% RSLogix 500 project TANK ANALOG CONTROL WITH ALARMS.RSS, saved by version 8.30.00.16 %
PROJECT "UNTITLED"    % processor: Bul.1763 MicroLogix 1100 Series B %

PROGRAM FILES
  LAD 2 "MAIN"  4 rungs
  LAD 3 "I/O"  5 rungs
  LAD 4 "CONTROLS"  6 rungs
  LAD 5 "ALARMS"  7 rungs

DATA FILES
  O0 OUTPUT  5 elements
  I1 INPUT  14 elements
  S2 STATUS  66 elements
  B3 BINARY  2 elements
  T4 TIMER  4 elements
  C5 COUNTER  1 elements
  R6 CONTROL  1 elements
  N7 INTEGER  1 elements
  F8 FLOAT  1 elements

LADDER 2 "MAIN"
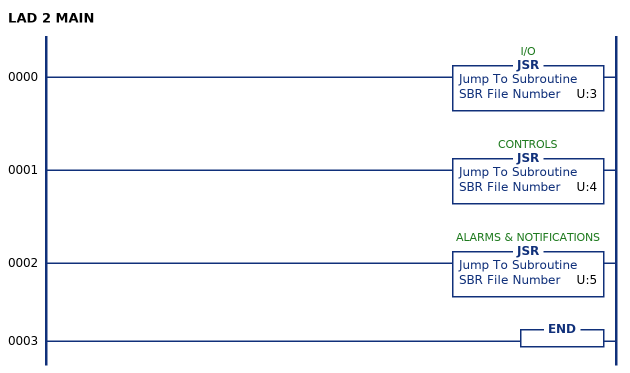
% Rung: 0 %
SOR JSR U:3 EOR
%   U:3  "I/O" %
% Rung: 1 %
SOR JSR U:4 EOR
%   U:4  "CONTROLS" %
% Rung: 2 %
SOR JSR U:5 EOR
%   U:5  "ALARMS & NOTIFICATIONS" %
% Rung: 3 %
SOR END EOR

LADDER 3 "I/O"
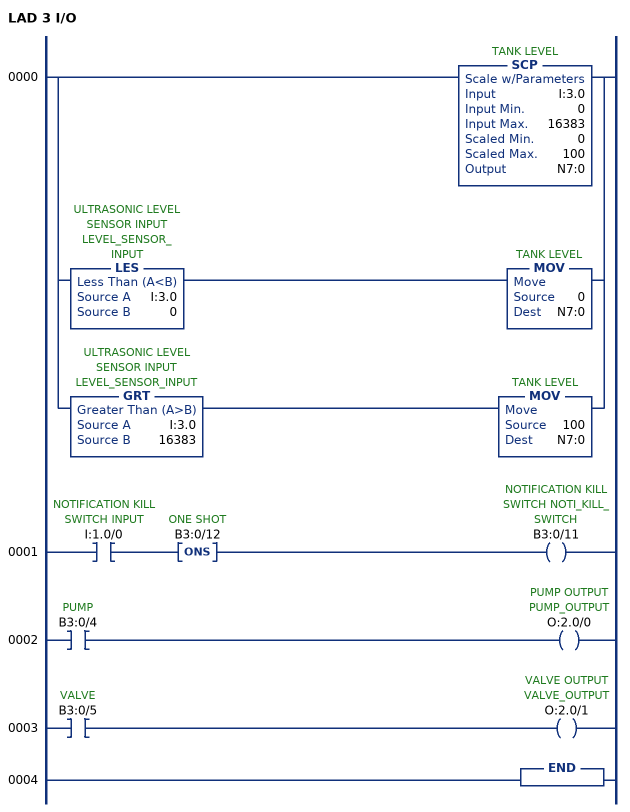
% Rung: 0 %
SOR BST SCP I:3.0 0 16383 0 100 N7:0 NXB LES I:3.0 0 MOV 0 N7:0 NXB GRT I:3.0 16383 MOV 100 N7:0 BND EOR
%   I:3.0  LEVEL_SENSOR_INPUT  "ULTRASONIC LEVEL SENSOR INPUT" %
%   N7:0  "TANK LEVEL" %
% Rung: 1 %
SOR XIC I:1.0/0 ONS B3:0/12 OTE B3:0/11 EOR
%   I:1.0/0  "NOTIFICATION KILL SWITCH INPUT" %
%   B3:0/12  "ONE SHOT" %
%   B3:0/11  NOTI_KILL_SWITCH  "NOTIFICATION KILL SWITCH" %
% Rung: 2 %
SOR XIC B3:0/4 OTE O:2.0/0 EOR
%   B3:0/4  "PUMP" %
%   O:2.0/0  PUMP_OUTPUT  "PUMP OUTPUT" %
% Rung: 3 %
SOR XIC B3:0/5 OTE O:2.0/1 EOR
%   B3:0/5  "VALVE" %
%   O:2.0/1  VALVE_OUTPUT  "VALVE OUTPUT" %
% Rung: 4 %
SOR END EOR

LADDER 4 "CONTROLS"
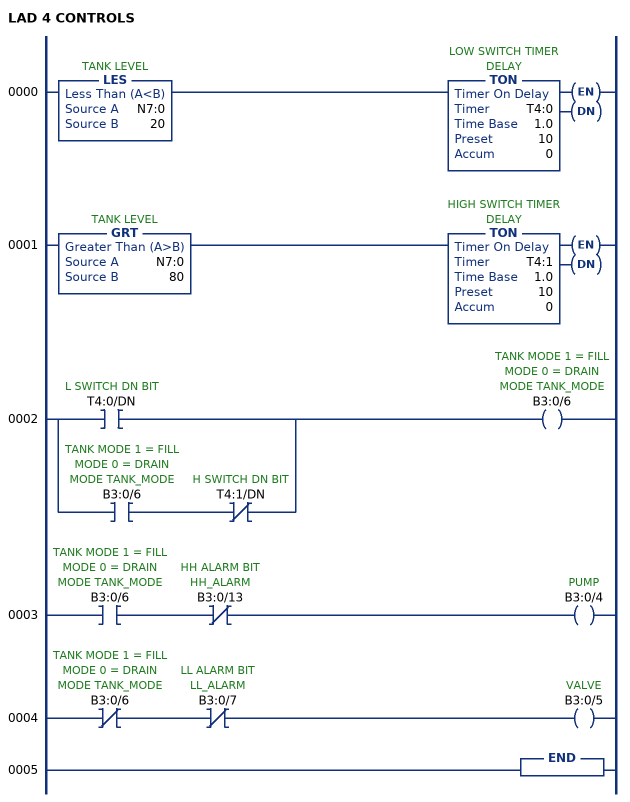
% Rung: 0 %
SOR LES N7:0 20 TON T4:0 1.0 10 0 EOR
%   N7:0  "TANK LEVEL" %
%   T4:0  "LOW SWITCH TIMER DELAY" %
% Rung: 1 %
SOR GRT N7:0 80 TON T4:1 1.0 10 0 EOR
%   N7:0  "TANK LEVEL" %
%   T4:1  "HIGH SWITCH TIMER DELAY" %
% Rung: 2 %
SOR BST XIC T4:0/DN NXB XIC B3:0/6 XIO T4:1/DN BND OTE B3:0/6 EOR
%   T4:0/DN  "L SWITCH DN BIT" %
%   B3:0/6  TANK_MODE  "TANK MODE 1 = FILL MODE 0 = DRAIN MODE" %
%   T4:1/DN  "H SWITCH DN BIT" %
% Rung: 3 %
SOR XIC B3:0/6 XIO B3:0/13 OTE B3:0/4 EOR
%   B3:0/6  TANK_MODE  "TANK MODE 1 = FILL MODE 0 = DRAIN MODE" %
%   B3:0/13  HH_ALARM  "HH ALARM BIT" %
%   B3:0/4  "PUMP" %
% Rung: 4 %
SOR XIO B3:0/6 XIO B3:0/7 OTE B3:0/5 EOR
%   B3:0/6  TANK_MODE  "TANK MODE 1 = FILL MODE 0 = DRAIN MODE" %
%   B3:0/7  LL_ALARM  "LL ALARM BIT" %
%   B3:0/5  "VALVE" %
% Rung: 5 %
SOR END EOR

LADDER 5 "ALARMS"
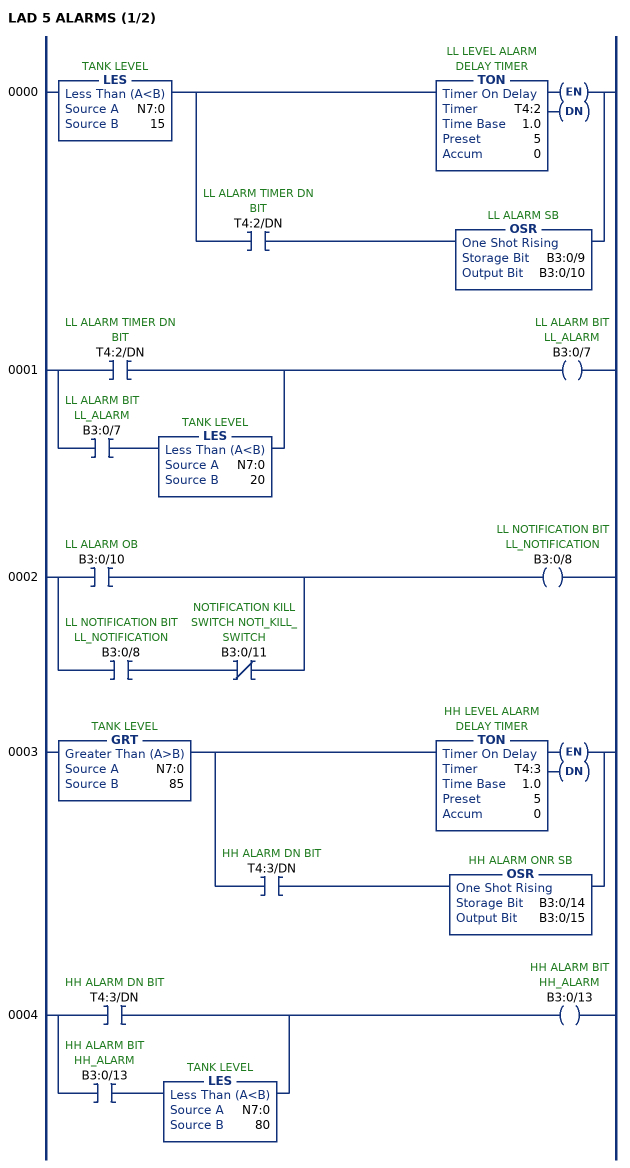
% Rung: 0 %
SOR LES N7:0 15 BST TON T4:2 1.0 5 0 NXB XIC T4:2/DN OSR B3:0/9 B3:0/10 BND EOR
%   N7:0  "TANK LEVEL" %
%   T4:2  "LL LEVEL ALARM DELAY TIMER" %
%   T4:2/DN  "LL ALARM TIMER DN BIT" %
%   B3:0/9  "LL ALARM SB" %
%   B3:0/10  "LL ALARM OB" %
% Rung: 1 %
SOR BST XIC T4:2/DN NXB XIC B3:0/7 LES N7:0 20 BND OTE B3:0/7 EOR
%   T4:2/DN  "LL ALARM TIMER DN BIT" %
%   B3:0/7  LL_ALARM  "LL ALARM BIT" %
%   N7:0  "TANK LEVEL" %
% Rung: 2 %
SOR BST XIC B3:0/10 NXB XIC B3:0/8 XIO B3:0/11 BND OTE B3:0/8 EOR
%   B3:0/10  "LL ALARM OB" %
%   B3:0/8  LL_NOTIFICATION  "LL NOTIFICATION BIT" %
%   B3:0/11  NOTI_KILL_SWITCH  "NOTIFICATION KILL SWITCH" %
% Rung: 3 %
SOR GRT N7:0 85 BST TON T4:3 1.0 5 0 NXB XIC T4:3/DN OSR B3:0/14 B3:0/15 BND EOR
%   N7:0  "TANK LEVEL" %
%   T4:3  "HH LEVEL ALARM DELAY TIMER" %
%   T4:3/DN  "HH ALARM DN BIT" %
%   B3:0/14  "HH ALARM ONR SB" %
%   B3:0/15  "HH ALARM ONS OB" %
% Rung: 4 %
SOR BST XIC T4:3/DN NXB XIC B3:0/13 LES N7:0 80 BND OTE B3:0/13 EOR
%   T4:3/DN  "HH ALARM DN BIT" %
%   B3:0/13  HH_ALARM  "HH ALARM BIT" %
%   N7:0  "TANK LEVEL" %

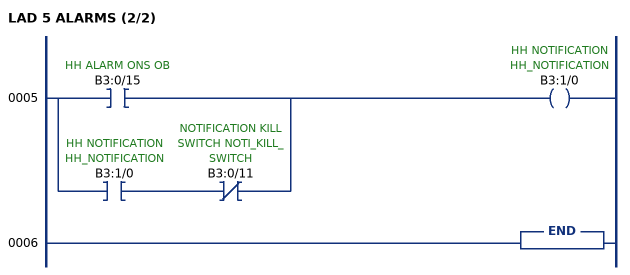
% Rung: 5 %
SOR BST XIC B3:0/15 NXB XIC B3:1/0 XIO B3:0/11 BND OTE B3:1/0 EOR
%   B3:0/15  "HH ALARM ONS OB" %
%   B3:1/0  HH_NOTIFICATION  "HH NOTIFICATION" %
%   B3:0/11  NOTI_KILL_SWITCH  "NOTIFICATION KILL SWITCH" %
% Rung: 6 %
SOR END EOR

OTHER DOCUMENTED ADDRESSES
  B3:0/0  LL_SWITCH_INPUT  "LL SWITCH INPUT"
  B3:0/1  L_SWITCH_INPUT  "L SWITCH INPUT"
  B3:0/2  H_SWITCH_INPUT  "H SWITCH INPUT"
  B3:0/3  HH_SWITCH_INPUT  "HH SWITCH INPUT"
  I:1.0/1  "L SWITCH"
  I:1.0/2  "H SWITCH"
  I:1.0/3  "HH SWITCH"

DATA TABLE (non-zero values as saved)
DATA T4
% .PRE .ACC %
% T4:0 % 10 0
% T4:1 % 10 0
% T4:2 % 5 0
% T4:3 % 5 0
